Universal Robots PolyScope program: OnRobot_Palletizing_Example.urp

Program OnRobot_Palletizing_Example (createdIn=3.3.1.237 lastSavedIn=3.7.0.40195 robotSerialNumber=2014359999 directory=/home/ur/ursim-current/programs/TransferVM/Examples/Pendrive installation=default)
Calibrated DH parameters: a=[0.000128, -0.175268, -0.306618, 0.000033, 0.000147, 0]; d=[0.089074, 542.39276, -475.591349, -66.691211, 0.094928, 0.082533]; alpha=[1.570044, -0.000714, -0.003663, 1.570304, -1.570247, 0]; deltaTheta=[0.000007, -1.145705, 0.472188, 0.673551, -0.000038, 0.000057]
BeforeStart
  URCap F/T Zero (FT-OnRobot, OnRobot A/S)
Robot Program (runOnlyOnce=false)
  MoveL speed 250 mm/s, acceleration 1200 mm/s^2 (useActiveTCP=false) feature=Base
    Waypoint PickWP: TCP in base x=-108.539 y=-431.763 z=146.072 mm, rx=-0.0012 ry=3.1163 rz=0.0389 rad; joints [-90.192, -98.598, -126.677, -46.161, 91.431, -0.254] deg
  'Insert your pick sequence.'
  URCap F/T Zero (FT-OnRobot, OnRobot A/S)
  URCap F/T Move (FT-OnRobot, OnRobot A/S) dataModel(speed=0.05, acceleration=0.5, coordsys=0, rpy=[0.0, 0.0, 0.0], popupLimit=false, ftarray=[0.0, 0.0, 0.0, 0.0, 0.0, 0.0, 0.0, 0.0], ftabsarray=[false, false, false, false, false, false], absolute=false)
    URCap F/T Waypoint (FT-OnRobot, OnRobot A/S) dataModel(relativeCoords=[0.0, 0.0, 0.07, 0.0, 0.0, 0.0], type=2, variable=pose_2, x=0.0, z=0.02)
  Pallet pattern(dimensionality=Box firstAxisCount=3 secondAxisCount=2 thirdAxisCount=2 motionType=MoveL speed=0.25 acceleration=1.2 useActiveTCP=false, counterVariable(name=cnt_2, initializeExpression=0), patternPoseVariable(name=pose_2), feature=Base, children(Waypoint(type=Fixed name=a1st_Corner_2, position(joints=-0.18179218126819663, -1.2063430807897628, -2.557153027115586, -0.949299738142301, 1.5693405272129537, 1.398648365020117 pose=0.32892438780945654, -0.2209372262081626, 0.17463595459184114, -1.3229276105014464E-4, -3.141587170192272, 5.6536918797502635E-5), poseInFeatureCoordinates=[0.328924, -0.220937, 0.174636, -0.000132, -3.141587, 0.000057], outputFlangePose=[0.328948, -0.220916, 0.274639, 0.000001, -3.141588, 0.000001]), Waypoint(type=Fixed name=a2nd_Corner_2, position(joints=-0.14819364287993153, -1.438525037908576, -2.4011777562769936, -0.8731015428759266, 1.5663272806089346, 1.432425213217349 pose=0.44593351045595736, -0.22512528078606533, 0.17461013611559537, -1.1469618927860493E-4, -3.1415675556745226, -1.0817243042016175E-5), poseInFeatureCoordinates=[0.445934, -0.225125, 0.17461, -0.000115, -3.141568, -0.000011], outputFlangePose=[0.445967, -0.225124, 0.274638, 0, -3.141588, 0.000001]), Waypoint(type=Fixed name=a3rd_Corner_2, position(joints=-0.027991817789214224, -1.386593807478878, -2.4419634710170497, -0.8842451952577797, 1.5670353672523571, 1.552617399408664 pose=0.44236491457327604, -0.16948484684153745, 0.1745704768802017, 1.2642847791794284E-4, -3.141355741998683, 2.5596207817989424E-5), poseInFeatureCoordinates=[0.442365, -0.169485, 0.17457, 0.000126, -3.141356, 0.000026], outputFlangePose=[0.442411, -0.169501, 0.274642, 0, -3.141588, 0.000001]), Waypoint(type=Fixed name=a4th_Corner_2, position(joints=-0.030268571576748116, -1.1351924597855714, -2.5924954997255476, -0.9851054719789261, 1.5701852497296453, 1.550050928400922 pose=0.33001392695138443, -0.16814049760643826, 0.17466593097346717, 2.959224207386941E-5, -3.141540530145319, 4.278931549116626E-5), poseInFeatureCoordinates=[0.330014, -0.16814, 0.174666, 0.00003, -3.141541, 0.000043], outputFlangePose=[0.330006, -0.168121, 0.274649, -0.000002, -3.141589, 0]), Waypoint(type=Fixed name=a5th_Corner_2, position(joints=-0.1926479793266651, -1.1327761322907008, -2.4845356593775056, -1.0954789816668686, 1.5698467515173693, 1.388387573483814 pose=0.32873636570711445, -0.22433458328272912, 0.22830374477111212, -7.668218169476655E-5, -3.141556107430171, -8.377758148491932E-5), poseInFeatureCoordinates=[0.328736, -0.224335, 0.228304, -0.000077, -3.141556, -0.000084], outputFlangePose=[0.328757, -0.224333, 0.328324, -0.000004, -3.141589, 0]), Waypoint(type=Fixed name=a6th_Corner_2, position(joints=-0.15871117085010056, -1.3533869922416528, -2.350483445047395, -1.0089300367460154, 1.5670227777593198, 1.42261139304979 pose=0.43821825605325004, -0.22856863429136132, 0.22838307996953253, 5.895732572495482E-5, 3.1414577714723975, -1.0110435115098015E-4), poseInFeatureCoordinates=[0.438218, -0.228569, 0.228383, 0.000059, 3.141458, -0.000101], outputFlangePose=[0.438186, -0.228542, 0.328337, -0.000006, -3.141589, 0]), Waypoint(type=Fixed name=a7th_Corner_2, position(joints=-0.02057031814105592, -1.310811904975182, -2.380536864084882, -1.0214497270070488, 1.567592187303191, 1.5607217517552439 pose=0.443927988088681, -0.16576590343260855, 0.22833551155381773, 9.627760541359413E-5, -3.1415720881706224, -1.7707389046682895E-5), poseInFeatureCoordinates=[0.443928, -0.165766, 0.228336, 0.000096, -3.141572, -0.000018], outputFlangePose=[0.443923, -0.165754, 0.328342, -0.000006, -3.141589, -0.000001]), Waypoint(type=Fixed name=a8th_Corner_2, position(joints=-0.025029871939679538, -1.048460384626427, -2.522676366961907, -1.1416505648993613, 1.5708427797787547, 1.5558179380491515 pose=0.3272961419784184, -0.16576960913939562, 0.22836130037851846, 1.1387693440751826E-4, -3.141555032183314, 1.5282244454355734E-4), poseInFeatureCoordinates=[0.327296, -0.16577, 0.228361, 0.000114, -3.141555, 0.000153], outputFlangePose=[0.327304, -0.165748, 0.328364, -0.000008, -3.141589, -0.000001]))); actionSequence(name=PalletSequence motionType=MoveL speed=0.25 acceleration=1.2 useActiveTCP=false, anchorWaypoint(type=Fixed name=PatternPoint_2, position(joints=-0.18276514886746043, -1.1515264400777987, -2.5112765130387005, -1.0499893103271063, 1.5697326568736383, 1.3980617258829113 pose=0.3289602808739009, -0.220907369224417, 0.21028219616628618, -6.134746356221756E-5, 3.141585898030077, -1.3132648306016172E-4), poseInFeatureCoordinates=[0.32896, -0.220907, 0.210282, -0.000061, 3.141586, -0.000131], outputFlangePose=[0.328942, -0.220906, 0.310252, 0.000001, -3.141587, 0.000002]), feature=Base, children(Waypoint(type=Fixed name=Approach_2, position(joints=-0.18450280776405137, -1.0837536119254212, -2.4264622053669105, -1.2025708489494722, 1.5702239912686466, 1.3969876086611377 pose=0.328952466789898, -0.22090074049658984, 0.27079575140169315, 6.998621950535503E-5, -3.1415346348778326, -7.928198650051173E-5), poseInFeatureCoordinates=[0.328952, -0.220901, 0.270796, 0.00007, -3.141535, -0.000079], outputFlangePose=[0.328947, -0.220908, 0.370782, 0.000001, -3.141588, 0.000002]), Waypoint=PatternPoint_2, Contributed(strategyProgramNodeType=F/T Search strategyURCapDeveloper=OnRobot A/S strategyURCapName=FT-OnRobot, dataModel(type=1, absolute=true, coordsys=1, speed=0.05, acceleration=0.5, rpy=[0.0, 0.0, 0.0], popupLimit=true, ftarray=[0.0, 0.0, 0.0, 0.0, 0.0, 0.0, 5.0, 0.1], ftabsarray=[false, false, false, false, false, false]), children(Contributed(strategyProgramNodeType=F/T Waypoint strategyURCapDeveloper=OnRobot A/S strategyURCapName=FT-OnRobot, dataModel(variable=pose_2, type=2, z=0.1)))), Comment(comment=Insert your place sequence.), Wait(type=Sleep, waitTime=1), Waypoint(type=Fixed name=Exit_2, position(joints=-0.18450194995324054, -1.0837739165632758, -2.426413363813921, -1.2026646731002995, 1.5702645779725395, 1.396944999743165 pose=0.3289572557322285, -0.22093915716177903, 0.27080577014899593, 9.925488335324977E-5, 3.1415700349272435, 3.835152960211542E-5), poseInFeatureCoordinates=[0.328957, -0.220939, 0.270806, 0.000099, 3.14157, 0.000038], outputFlangePose=[0.328958, -0.220906, 0.370796, 0.00007, -3.141535, -0.000079])))
    Pattern -> pattern
    AnchoredSequence -> PalletSequence
